TYPE Icon :
STRUCT
	Title : STRING;
	IconType : STRING;
	Signal : BOOL;
	BlinkingEnabled : BOOL := FALSE;
	EnableRedIcon : BOOL := TRUE;
	
	///used internally
	SignalBlink : BOOL;
END_STRUCT
END_TYPE

(* stored: Version 1.1.0.1
   DUT Icon: Id {a5ceab7d-2229-477d-b701-571013b76bf8} *)
